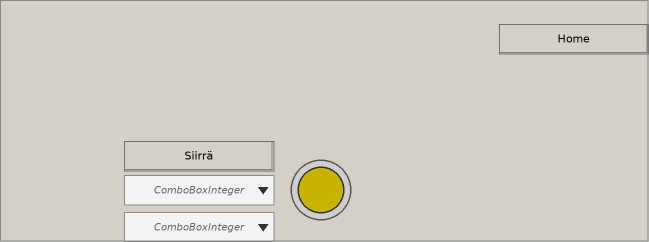
VISUALIZATION Visualization  // 649x242
    Button (499,24 150x30), "Home"
        tap Comms.kotiutusnappi
    Lamp1 (286,155 70x70), style: Lamp-Lamp1-Yellow
    ComboBoxInteger (124,212 150x30), variable: Comms.stSlotCmd.to_slot
    Button (124,141 150x30), "Siirrä"
        tap Comms.bSlotCmd
    ComboBoxInteger (124,175 150x30), variable: Comms.stSlotCmd.from_slot
END_VISUALIZATION

(* stored: Version 1.1.0.1, ProductVersion 3.1.4024.12
   Visu Visualization: Id {47d02903-534e-479a-a5c4-bd1c47095a15} *)
